Fanuc KAREL source: kt00412.KL

-- PROVISIONAL review KL for V940-1; original PC SHA256 158443985f4cbbf9243d3a71a8804f1f7b3002a5c9f9f7de12e69706ddee0df4
-- Incomplete behavior may be omitted. Consult companion uncertainty JSON. Do not deploy.
PROGRAM KT00412
%NOLOCKGROUP
VAR
  R2 : REAL
  OUT : BOOLEAN
-- UNRESOLVED_DECL Y1 type=002018
BEGIN
  -- V9_ZERO_TABLE_METADATA_HINT layout=0001; no indexed target words; source/name/runtime held
  -- UNRESOLVED_PC offsets 5-19; opcodes 2E,22,9D,33,B2
  -- UNRESOLVED_PC offsets 24-35; opcodes 2E,23
  -- UNRESOLVED_PC offsets 40-65; opcodes 22,9D,33,B1,21,29,64,29,71,23
  -- UNRESOLVED_PC offsets 70-74; opcodes 7F
END KT00412
